(* IEC 61131-3 sources: OpenPLC_Sample_Programs/st-checker/ST_Tests, 3 files *)

(* ---- input2.st ---- *)
FUNCTION_BLOCK MaxMin
VAR_INPUT
	T_Inputs : ARRAY [1..5] OF REAL;
END_VAR
VAR
	i: INT:=1;
END_VAR
VAR_OUTPUT
	MAXnum : REAL := 0.0;
	MINnum : REAL := 2000.0;
END_VAR

WHILE i<=5 DO
	IF T_Inputs[i] > MAXNum
		THEN MAXnum := T_Inputs[i];
	END_IF;
	IF T_Inputs[i] < MinNum
		THEN Minnum := T_Inputs[i];
	END_IF;
	i := i+1;
END_WHILE;

END_FUNCTION_BLOCK

PROGRAM Main
VAR
	PP : MaxMin;
	i: INT:=1;
END_VAR
VAR_OUTPUT
	MAXnum : REAL;
	MINnum : REAL;
END_VAR
VAR_INPUT
	T_Inputs1 : ARRAY [1..5] OF REAL;
END_VAR

(* PP(T_Inputs:=T_Inputs1); *)
WHILE i<=5 DO
	PP.T_Inputs[1] := T_Inputs1[i];
	i := i+1;
END_WHILE;

MAXnum := PP.MAXnum;
MINnum := PP.MINnum;

END_PROGRAM

CONFIGURATION Config0
  RESOURCE Res0 ON PLC
    TASK task0(INTERVAL := T#50ms, PRIORITY := 0);
    PROGRAM instance0 WITH task0 : Main;
  END_RESOURCE
END_CONFIGURATION

(* ---- fibonacci-numbers.st ---- *)
FUNCTION AddTwo : INT
  VAR_INPUT
    In0 : INT;
    In1 : INT;
  END_VAR
  AddTwo := In0 + In1;
END_FUNCTION

PROGRAM program0
  VAR_INPUT
    N : INT := 5;
  END_VAR
  VAR_OUTPUT
    O : INT := 1;
  END_VAR
  VAR
    F1 : INT := 1;
    F2 : INT := 1;
    CNT : INT := 2;
  END_VAR

  IF N <= CNT THEN
    O := 1;
  ELSE
    WHILE CNT < N DO
      O := AddTwo(In0:=F1, In1:=F2);
      F1 := F2;
      F2 := O;
      CNT := CNT + 1;
    END_WHILE;
  END_IF;
END_PROGRAM

CONFIGURATION Config0
  RESOURCE Res0 ON PLC
    TASK task0(INTERVAL := T#50ms, PRIORITY := 0);
    PROGRAM instance0 WITH task0 : program0;
  END_RESOURCE
END_CONFIGURATION

(* ---- input.st ---- *)
FUNCTION increment : int
    VAR_INPUT
        in0, in1 : INT;
    END_VAR
    VAR
        test : INT := 10;
        ba : BOOL;
    END_VAR
    VAR_OUTPUT
        out : INT;
    END_VAR

    out := in0 + in1;
    increment := out;
END_FUNCTION

PROGRAM Main
VAR_INPUT
    IN, IN1 : INT;
    IN2 : INT := 10;
END_VAR
VAR_TEMP
    CNT : INT;
    F1, F2 : INT;
END_VAR
VAR_OUTPUT
    OUT : INT;
END_VAR

IF IN < 3 THEN
    OUT := 1;
ELSE
    WHILE CNT < IN DO
        OUT := increment(in0 := F1, in1 := F2, out => OUT) + 1;
        F1 := F2;
        F2 := OUT;
        CNT := CNT + 1;
    END_WHILE;
END_IF;

END_PROGRAM

CONFIGURATION Config0
  RESOURCE Res0 ON PLC
    TASK task0(INTERVAL := T#50ms, PRIORITY := 0);
    PROGRAM instance0 WITH task0 : Main;
  END_RESOURCE
END_CONFIGURATION
